PROGRAM DbWriteInfluxDB
VAR
	// Cycle record data
	fbInfluxDBRecorder	:RecordInfluxDB;
END_VAR

// Insert DB
fbInfluxDBRecorder(
	command_queue := GVL.tsdb_command_queue,
	nDBID := 1      // Database ID by TF6420 configurator
);

END_PROGRAM

(* stored: Version 1.1.0.1, ProductVersion 3.1.4024.12
   POU DbWriteInfluxDB: Id {b3c9b1c0-8e19-46d8-955e-27b35c8007f9}, SpecialFunc None *)
